{attribute addProperty BoxType "IODEVICETYPE_ETHERCATPROT"}
{attribute addProperty Id "Beckhoff_EK11xxBeckhoff_EK11xx_69A876EE56070Beckhoff_EK12xxBeckhoff_EK12xx_26FD3E4A162Beckhoff_EK13xxBeckhoff_EK13xx_81521E8116020Beckhoff_EK15xxBeckhoff_EK15xx_DE996DDF76896Beckhoff_EK18xxBeckhoff_EK18xx_11305A3F1432179Beckhoff_EKM1xxxBeckhoff_EKM1xxx_21EDF19F2971371.375Beckhoff_EKx9xxBeckhoff_EKx9xx_CA467E2B4688586Beckhoff_EKxxxx_0080Beckhoff_EKxxxx_0080_F8E2E0BC648SyncUnitsSyncUnits_3FA29F3C21627InputsInputs_C75D3FEC1280160OutputsOutputs_47D1E803848106InfoDataInfoData_45F98C5022428"}
{attribute addProperty CRC "1669166991"}
{attribute addProperty SizeInBites "13227"}
{attribute addProperty SizeInBytes "1653.375"}
TYPE EtherCAT_Master_EKxxxx_637D778F :
STRUCT
	{attribute addProperty Name "Beckhoff_EK11xx"}
	Beckhoff_EK11xx : Beckhoff_EK11xx_69A876EE;
	{attribute addProperty Name "Beckhoff_EK12xx"}
	Beckhoff_EK12xx : Beckhoff_EK12xx_26FD3E4A;
	{attribute addProperty Name "Beckhoff_EK13xx"}
	Beckhoff_EK13xx : Beckhoff_EK13xx_81521E81;
	{attribute addProperty Name "Beckhoff_EK15xx"}
	Beckhoff_EK15xx : Beckhoff_EK15xx_DE996DDF;
	{attribute addProperty Name "Beckhoff_EK18xx"}
	Beckhoff_EK18xx : Beckhoff_EK18xx_11305A3F;
	{attribute addProperty Name "Beckhoff_EKM1xxx"}
	Beckhoff_EKM1xxx : Beckhoff_EKM1xxx_21EDF19F;
	{attribute addProperty Name "Beckhoff_EKx9xx"}
	Beckhoff_EKx9xx : Beckhoff_EKx9xx_CA467E2B;
	{attribute addProperty Name "Beckhoff_EKxxxx_0080"}
	Beckhoff_EKxxxx_0080 : Beckhoff_EKxxxx_0080_F8E2E0BC;
	{attribute addProperty Name "SyncUnits"}
	SyncUnits : SyncUnits_3FA29F3C;
	{attribute addProperty Name "Inputs"}
	Inputs : Inputs_C75D3FEC;
	{attribute addProperty Name "Outputs"}
	Outputs : Outputs_47D1E803;
	{attribute addProperty Name "InfoData"}
	InfoData : InfoData_45F98C50;
END_STRUCT
END_TYPE

(* stored: Version 1.2.0.0, ProductVersion 3.1.4024.9
   DUT EtherCAT_Master_EKxxxx_637D778F: Id {e0c112d8-8214-442a-ac85-66b5e58398c4} *)
